
FUNCTION CB_word_to_dint : DINT

TITLE = ' Convert a word into a Double integer '
VERSION : '1.0'
AUTHOR  : CB
NAME    : DworToDi
FAMILY  : TNI

VAR_INPUT
    IN : WORD;
END_VAR

VAR_TEMP

END_VAR

BEGIN

CB_word_to_dint := WORD_TO_DINT(IN);

END_FUNCTION
